FUNCTION_BLOCK Station001 EXTENDS TcoCore.TcoContext
VAR
	
	{attribute addProperty Name "Long running example"}
	LongRunningTask : TcoCore.TcoTask(THIS^, NO.Structure);
	i :int;
	_components : Station001_Components(THIS^, NO.Structure);
	
	_sequence : Station001_Sequencer(THIS^, NO.Structure, eRestoreMode.None, _components);
END_VAR

(*~
	<docu>
		<summary>
			Main method of the TcoContext. This is the entry point of any control logic that belongs to this context. 
			The call of this method is ensured by calling the <c>InstanceName.Run()</c> method, and it must not be called explicitly.
			This method is abstract, and it must be overridden in derived block.
		</summary>
	</docu>
~*)
METHOD PROTECTED  Main
_sequence.Run();

IF(LongRunningTask.Execute()) THEN
	i:= i+1;
	IF(i MOD 2000 = 0)THEN
		i:=1;
		LongRunningTask.DoneWhen(TRUE);
	END_IF
END_IF
END_METHOD

END_FUNCTION_BLOCK

(* stored: Version 1.1.0.1
   POU Station001: Id {52997647-59b7-0080-2171-dd40855e4ef4}, SpecialFunc None
   Method Main: Id {81d16536-e5af-00c3-2280-eeb002086c65} *)
